(* IEC 61131-3 sources: CannyIEC/extracted_st/cannyiec/functions/rsignbit, 1 file *)

(* ---- RSIGNBIT.st ---- *)
(* --- Interface --- *)
FUNCTION RSIGNBIT : BIT
VAR_INPUT
    rValue : REAL;
END_VAR
(* --- Implementation --- *)
RSIGNBIT := rValue < REAL#0;
